FUNCTION_BLOCK Multiplex
VAR_INPUT
	In1: BOOL;
	In2: BOOL;
	In3: BOOL;
END_VAR
VAR_OUTPUT
	Out1: BOOL;
	Out2: BOOL;
	Out3: BOOL;
	Out4: BOOL;
END_VAR
VAR
	RS_1: RS;
	RS_2: RS;
	RS_3: RS;
	RS_5: RS;
	TON_4: TON;
	TON_3: TON;
	TON_2: TON;
	TON_1: TON;
END_VAR

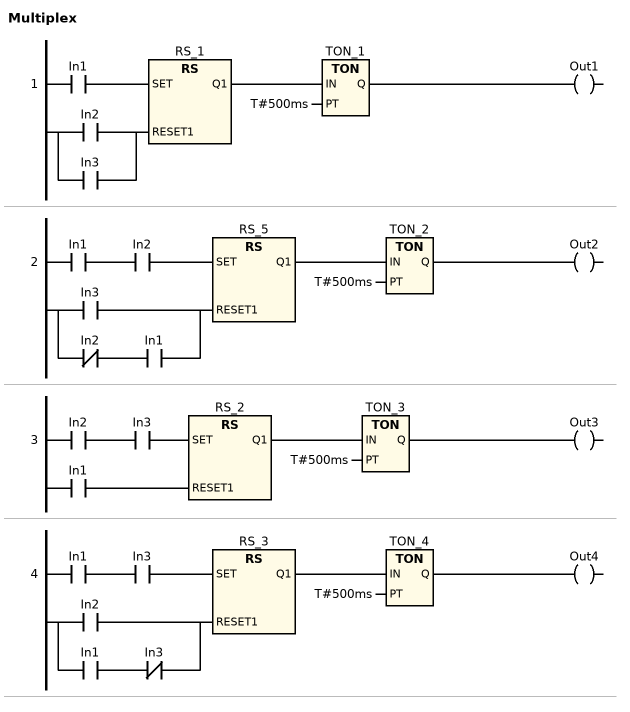
// NETWORK 1
RS_1(SET := In1, RESET1 := In2 OR In3); // RS
TON_1(IN := RS_1.Q1, PT := T#500ms); // TON
Out1 := TON_1.Q;

// NETWORK 2
RS_5(SET := In1 AND In2, RESET1 := In3 OR NOT In2 AND In1); // RS
TON_2(IN := RS_5.Q1, PT := T#500ms); // TON
Out2 := TON_2.Q;

// NETWORK 3
RS_2(SET := In2 AND In3, RESET1 := In1); // RS
TON_3(IN := RS_2.Q1, PT := T#500ms); // TON
Out3 := TON_3.Q;

// NETWORK 4
RS_3(SET := In1 AND In3, RESET1 := In2 OR In1 AND NOT In3); // RS
TON_4(IN := RS_3.Q1, PT := T#500ms); // TON
Out4 := TON_4.Q;

END_FUNCTION_BLOCK

(* stored: Version 1.1.0.1, ProductVersion 3.1.4024.12
   POU Multiplex: Id {57a65343-f85f-4f6f-b8d0-e33227bef4c2}, SpecialFunc None *)
